// TwinCAT 3 PLC project StateStation
// ProgramVersion: 3.1.4023.0
// libraries:
//   Tc2_Standard, * (Beckhoff Automation GmbH)
//   Tc2_System, * (Beckhoff Automation GmbH)
//   Tc3_Module, * (Beckhoff Automation GmbH)
// project tree:
//   DUTs/ FB_BaseState.TcPOU, FB_State_Idle.TcPOU, FB_Stattion.TcPOU, Istate.TcIO
//   / PlcTask.TcTTO
//   POUs/ MAIN.TcPOU
// real-time tasks:
//   TASK PlcTask: cycle T#10ms, priority 20, ADS port 350

CONFIGURATION StateStation
    RESOURCE PLC ON TwinCAT3
        TASK PlcTask(INTERVAL := T#10ms, PRIORITY := 20);
        PROGRAM MAIN WITH PlcTask : MAIN;
    END_RESOURCE
END_CONFIGURATION

// ---- DUTs/Istate.TcIO
INTERFACE Istate

METHOD mExecute
VAR_INPUT
END_VAR
END_METHOD

METHOD mHold
VAR_INPUT
END_VAR
END_METHOD

METHOD mStart
VAR_INPUT
END_VAR
END_METHOD

METHOD mStop
VAR_INPUT
END_VAR
END_METHOD

PROPERTY pMessage : String
GET
END_GET
END_PROPERTY

END_INTERFACE

// ---- POUs/MAIN.TcPOU
PROGRAM MAIN
VAR
END_VAR

END_PROGRAM

// ---- DUTs/FB_BaseState.TcPOU
FUNCTION_BLOCK FB_BaseState IMPLEMENTS Istate
VAR_INPUT
END_VAR
VAR_OUTPUT
END_VAR
VAR
	_pStation		: REFERENCE TO FB_Station;
	bIsInitalized	: BOOL;
END_VAR

METHOD FB_init : BOOL
VAR_INPUT
	bInitRetains : BOOL; // if TRUE, the retain variables are initialized (warm start / cold start)
	bInCopyCode : BOOL;  // if TRUE, the instance afterwards gets moved into the copy code (online change)
	
	StationPointer 	: POINTER TO FB_Station;
END_VAR
END_METHOD

{warning 'add method implementation '}
METHOD mExecute
END_METHOD

{warning 'add method implementation '}
METHOD mHold
END_METHOD

{warning 'add method implementation '}
METHOD mStart
END_METHOD

{warning 'add method implementation '}
METHOD mStop
END_METHOD

PROPERTY pMessage : STRING
GET
END_GET
END_PROPERTY

{attribute 'monitoring' := 'variable'}
PROPERTY pStation : REFERENCE TO FB_Station;
GET
pStation REF= _pStation;
END_GET
SET
_pStation REF= pStation;
END_SET
END_PROPERTY

END_FUNCTION_BLOCK

// ---- DUTs/FB_State_Idle.TcPOU
FUNCTION_BLOCK FB_State_Idle EXTENDS FB_BaseState IMPLEMENTS Istate
VAR_INPUT
END_VAR
VAR_OUTPUT
END_VAR
VAR
END_VAR

METHOD mStart
ADSLOGSTR(ADSLOG_MSGTYPE_HINT, 'Start signal asserted.', '');
END_METHOD

{error 'add property implementation or delete property to use base implementation'}
PROPERTY pMessage : STRING
GET
pMessage := 'Waiting for start signal';
END_GET
END_PROPERTY

END_FUNCTION_BLOCK

// ---- DUTs/FB_Stattion.TcPOU
FUNCTION_BLOCK FB_Stattion
VAR_INPUT
	bStart				: BOOL;
	bStop				: BOOL;
	bHold				: BOOL;
END_VAR
VAR_OUTPUT
	iCurrentState		: Istate := fbStateIdle;
END_VAR
VAR
	fbStateIdle			: FB_State_Idle(THIS);
END_VAR

END_FUNCTION_BLOCK
